INTERFACE I_UnitTestResultFile EXTENDS __SYSTEM.IQueryInterface

METHOD AddTestCaseResult
VAR_INPUT
	TestClassName	: STRING;
	TestName		: STRING;
	Duration		: LREAL;
	FailureMessage : STRING := '';
	FailureType	: STRING := '';
	FailureNote	: STRING := '';
END_VAR
END_METHOD

METHOD AddTestSuite
VAR_INPUT
	Name	  : STRING;
END_VAR
END_METHOD

METHOD AddTestSuiteStatistics
VAR_INPUT
	Name	  : STRING;
	Tests	  : UDINT;
	Failures : UDINT := 0;
	Errors	  : UDINT := 0;
	Skipped	  : UDINT := 0;
	Duration  : LREAL;
END_VAR
END_METHOD

METHOD Cyclic
VAR_INPUT
END_VAR
END_METHOD

METHOD Initialize
VAR_INPUT
	ReInitialize : BOOL := FALSE;
END_VAR
END_METHOD

{attribute 'monitoring' := 'call'}
PROPERTY Initialized : BOOL
GET
END_GET
END_PROPERTY

{attribute 'monitoring' := 'call'}
PROPERTY Path : STRING
SET
END_SET
END_PROPERTY

METHOD SaveResult
VAR_INPUT
END_VAR
END_METHOD

END_INTERFACE

(* stored: Version 1.1.0.1
   Itf I_UnitTestResultFile: Id {e1366dc8-517e-46ad-b1e3-80eafaf62fca}
   Method AddTestCaseResult: Id {3b1e675c-601a-4597-82c3-21011f29cf49}
   Method AddTestSuite: Id {336643ed-f4f2-4062-ab5f-cbc7284ffffe}
   Method AddTestSuiteStatistics: Id {ab144702-dfd4-4808-ac97-0c41b9b09781}
   Method Cyclic: Id {498d2274-e054-4c85-ba80-3f227ed28def}
   Method Initialize: Id {7c254bb1-9728-4958-adfe-eece97237b3f}
   Property Initialized: Id {13066041-fb66-4ac5-8cb1-564d985f7edb}
   Get Get: Id {214d7296-ccd6-4e4b-b4db-c68a08bccd9f}
   Property Path: Id {d5e878b1-73ea-46b7-af48-f47146e27775}
   Set Set: Id {6d62ca58-efa1-4260-80f9-2e1c1e497795}
   Method SaveResult: Id {690c3506-9c68-4a55-8088-e8b719c43680} *)
